Staubli VAL3: OnEvent6.pgx

program OnEvent6()
begin
  //-----------------------------------------------------------------------
  //Header begin
  //LasMAN3.7
  //Description of program
  //
  //Input parameters
  //
  //Output paramaters
  //Example
  //  call OnEvent1()
  //History
  //  Creation : 2013-06-23  y.ye@staubli.com
  //Header end
  //-----------------------------------------------------------------------
  if DataBase:nRemoteProduct==8888
    call Teach:TeachRemote()
  else
    popUpMsg("远程生产密码不正确")
  endIf
  DataBase:nInterfaceType=9
end
